TYPE _ST_ERROR_ :
STRUCT
	CODE 	: INT;
	SOURCE 	: STRING(255);
	STATUS 	: BOOL;
END_STRUCT
END_TYPE

(* stored: Version 1.1.0.1, ProductVersion 3.1.4022.18
   DUT _ST_ERROR_: Id {8f8f9496-fce9-4bb0-b8ee-f9ba713f7871} *)
